(* IEC 61131-3 sources: RAG_PLC/data/result/test/004, 2 files *)

(* ---- wrapped.st ---- *)
(* =========================================================
   Generated by PLC-Eval Benchmark Wrapper
   ========================================================= *)

FUNCTION_BLOCK LLM_Wrapper_FB
VAR_INPUT
	STR : STRING;
END_VAR

VAR_OUTPUT
	CAPITALIZE : STRING;
END_VAR

VAR
	char : BYTE;
	char2 : BYTE;
	pos : INT;
	L : INT;
	first : BOOL;
	str_temp : STRING;
END_VAR

CAPITALIZE := STR;
first := TRUE;
L := LEN(STR);
FOR pos := 1 TO L DO
	char := INT_TO_BYTE(GET_CHAR(STR, pos));
	IF first THEN
		char2 := TO_UPPER(char);
		IF char <> char2 THEN
			str_temp := CAPITALIZE;
			CAPITALIZE := REPLACE(str_temp, BYTE_TO_STRING(char2, '%c'), 1, pos);
		END_IF;
	END_IF;
	(* 记住下一个字符是否需要大写 *)
	first := char = BYTE#32;
END_FOR;
END_FUNCTION_BLOCK

PROGRAM Auto_Proxy_Prg
  VAR
    instance : LLM_Wrapper_FB;
  END_VAR

  instance();
END_PROGRAM

CONFIGURATION Config0
  RESOURCE Res0 ON PLC
    TASK TaskMain(INTERVAL := T#20ms, PRIORITY := 0);
    PROGRAM Inst0 WITH TaskMain : Auto_Proxy_Prg;
  END_RESOURCE
END_CONFIGURATION

(* ---- raw_code.st ---- *)
VAR_INPUT
	STR : STRING;
END_VAR

VAR_OUTPUT
	CAPITALIZE : STRING;
END_VAR

VAR
	char : BYTE;
	char2 : BYTE;
	pos : INT;
	L : INT;
	first : BOOL;
	str_temp : STRING;
END_VAR

CAPITALIZE := STR;
first := TRUE;
L := LEN(STR);
FOR pos := 1 TO L DO
	char := INT_TO_BYTE(GET_CHAR(STR, pos));
	IF first THEN
		char2 := TO_UPPER(char);
		IF char <> char2 THEN
			str_temp := CAPITALIZE;
			CAPITALIZE := REPLACE(str_temp, BYTE_TO_STRING(char2, '%c'), 1, pos);
		END_IF;
	END_IF;
	(* 记住下一个字符是否需要大写 *)
	first := char = BYTE#32;
END_FOR;
